(* CoDeSys 2.3 project: drillMachine_Simple_Turku.pro *)
(* Title: Use of different IEC-61131-3 languages *)
(* Version: 1.0.0 *)
(* Author: Niko Siltala (TUT) *)
(* Description: Use of different IEC-61131-3 languages to control a lift door. *)
(* Libraries: Util.lib 16.8.17 14:08:57, STANDARD.LIB 16.8.17 14:08:57 *)

(* Global variable list: Global_Variables *)
VAR_GLOBAL
	(*ConveyourIn - Left*)
	I_ConvIn_PartPresent: BOOL;	(*Sensor: Part is present*)
	O_ConvIn_MotON		: BOOL;	(*Conveyour In: Motor ON*)

	(*ConveyourOut - Right*)
	I_ConvOut_PartPresent: BOOL;(*Sensor: Part is present*)
	O_ConvOut_MotON		: BOOL;	(*Conveyour Out: Motor ON*)

	(*Manipulator - Left*)
	I_ManiL_Limit_Up	: BOOL;	(*Manipulator Left: Limit: Up*)
	I_ManiL_Limit_Dn	: BOOL;	(*Manipulator Left: Limit: Down*)
	I_ManiL_Limit_Home	: BOOL;	(*Manipulator Left: Home sensor*)
	I_ManiL_Turned_Left	: BOOL;	(*Manipulator Left: Turned to left*)
	I_ManiL_Turned_Right: BOOL;	(*Manipulator Left: Turned to right*)
	I_ManiL_Gripper_Open: BOOL;	(*Manipulator Left: Gripper is open*)

	O_ManiL_Turn_Left	: BOOL;	(*Manipulator Left: Turn to left position. Controls the valve*)
	O_ManiL_Turn_Right	: BOOL;	(*Manipulator Left: Turn to right position. Controls the valve*)
	O_ManiL_Gripper_Close: BOOL;(*Manipulator Left: Closes Gripper. Controls the valve*)

	bManiL_axZ_Enable	: BOOL;	(*Manipulator Left: Z-axis: enable*)
	bManiL_axZ_Start	: BOOL;	(*Manipulator Left: Z-axis: Start motion*)
	fManiL_axZ_Velo		: REAL;	(*Manipulator Left: Z-axis: Velocity*)
	fManiL_axZ_TargetPos: REAL;	(*Manipulator Left: Z-axis: Target position*)
	fManiL_axZ_CurrPos	: REAL;	(*Manipulator Left: Z-axis: Current position*)
	bManiL_axZ_InTargetPos	: BOOL;	(*Manipulator Left: Z-axis: Target position is reached*)

	(*Drilling Machine*)
	I_Drill_Limit_Up	: BOOL;	(*Drill: Limit: Up*)
	I_Drill_Limit_Dn	: BOOL;	(*Drill: Limit: Down*)
	I_Drill_Limit_Home	: BOOL;	(*Drill: Home sensor*)
	I_Drill_Fixture_Open: BOOL;	(*Drill: Fixture is open*)
	I_Drill_Fixture_Closed: BOOL;	(*Drill: Fixture is closed*)

	O_Drill_Spindle_On	: BOOL;	(*Drill: Turn on drill spindle.*)
	O_Drill_Fixture_Close: BOOL;(*Drill: Closes Fixture. Controls the valve*)

	bDrill_axZ_Enable	: BOOL;	(*Drill: Z-axis: enable*)
	bDrill_axZ_Start	: BOOL;	(*Drill: Z-axis: Start motion*)
	fDrill_axZ_Velo		: REAL;	(*Drill: Z-axis: Velocity*)
	fDrill_axZ_TargetPos: REAL;	(*Drill: Z-axis: Target position*)
	fDrill_axZ_CurrPos	: REAL;	(*Drill: Z-axis: Current position*)
	bDrill_axZ_InTargetPos	: BOOL;	(*Drill: Z-axis: Target position is reached*)

	(*Manipulator - Right*)
	I_ManiR_Limit_Up	: BOOL;	(*Manipulator Right: Limit: Up*)
	I_ManiR_Limit_Dn	: BOOL;	(*Manipulator Right: Limit: Down*)
	I_ManiR_Limit_Home	: BOOL;	(*Manipulator Right: Home sensor*)
	I_ManiR_Turned_Left	: BOOL;	(*Manipulator Right: Turned to left*)
	I_ManiR_Turned_Right: BOOL;	(*Manipulator Right: Turned to right*)
	I_ManiR_Gripper_Open: BOOL;	(*Manipulator Right: Gripper is open*)

	O_ManiR_Turn_Left	: BOOL;	(*Manipulator Right: Turn to left position. Controls the valve*)
	O_ManiR_Turn_Right	: BOOL;	(*Manipulator Right: Turn to right position. Controls the valve*)
	O_ManiR_Gripper_Close: BOOL;(*Manipulator Right: Closes Gripper. Controls the valve*)

	bManiR_axZ_Enable	: BOOL;	(*Manipulator Right: Z-axis: enable*)
	bManiR_axZ_Start	: BOOL;	(*Manipulator Right: Z-axis: Start motion*)
	fManiR_axZ_Velo		: REAL;	(*Manipulator Right: Z-axis: Velocity*)
	fManiR_axZ_TargetPos: REAL;	(*Manipulator Right: Z-axis: Target position*)
	fManiR_axZ_CurrPos	: REAL;	(*Manipulator Right: Z-axis: Current position*)
	bManiR_axZ_InTargetPos	: BOOL;	(*Manipulator Right: Z-axis: Target position is reached*)


	(*Control panel and indications*)
	I_EmergencyClear	: BOOL;	(*Emergency Circuit is clear*)
	I_Btn_Reset		: BOOL;	(*Button: Reset*)
	I_Btn_Start		: BOOL;	(*Button: Start*)
	I_Btn_Stop		: BOOL;	(*Button: Stop*)
	I_Btn_CycleStart: BOOL;	(*Button: Cycle Start*)

	O_Light_Running	: BOOL;	(*Light: Running*)
	O_Light_Stopped	: BOOL;	(*Light: Stopped*)
	O_Beacon_Red	: BOOL;	(*Beacon Light: red*)
	O_Beacon_Yellow	: BOOL;	(*Beacon Light: yellow*)
	O_Beacon_Green	: BOOL;	(*Beacon Light: green*)

END_VAR

(* Data type *)
TYPE ST_Part :
(*Data structure for the simulated parts *)
STRUCT
	bExists		: BOOL;	(* Part exists *)
	bHasHole	: BOOL;	(* Part has hole *)
	posX		: REAL;	(* X-position of the part*)
	posY		: REAL;	(* Y-position of the part*)
END_STRUCT
END_TYPE

(* POU PRG_MAIN, ST *)
PROGRAM PRG_MAIN
VAR
	fbSFCExample : FB_SFC_Example;
END_VAR
(*START MAKING YOUR DRILLING SYSTEM PROGRAM HERE*)
fbSFCExample();
PRG_SFCDrilling(bReset:= );
END_PROGRAM

(* POU Examples/FB_SFC_Example, SFC *)
FUNCTION_BLOCK FB_SFC_Example
VAR_INPUT
	bReset		: BOOL;	(*Reset Request*)
END_VAR
VAR_OUTPUT
END_VAR
VAR
	bLocalReset	: BOOL;	(*Performs local reset*)
	SFCReset 	: BOOL;	(*Resets the execution of SFC to init once this SFCFlag is set true *)
END_VAR
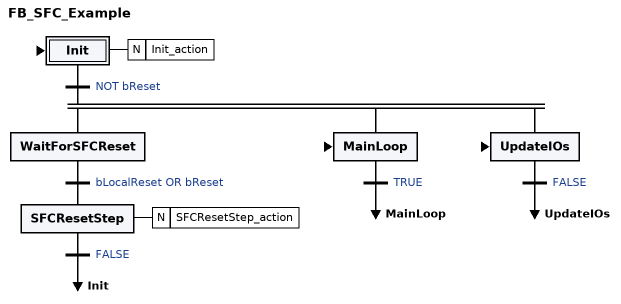
INITIAL_STEP Init:
	Init_action(N);
END_STEP
TRANSITION FROM Init TO (WaitForSFCReset, MainLoop, UpdateIOs) := NOT bReset;
END_TRANSITION
STEP WaitForSFCReset:
END_STEP
TRANSITION FROM WaitForSFCReset TO SFCResetStep := bLocalReset OR bReset;
END_TRANSITION
STEP SFCResetStep:
	SFCResetStep_action(N);
END_STEP
TRANSITION FROM SFCResetStep TO Init := FALSE;
END_TRANSITION
STEP MainLoop:
END_STEP
TRANSITION FROM MainLoop TO MainLoop := TRUE;
END_TRANSITION
STEP UpdateIOs:
END_STEP
TRANSITION FROM UpdateIOs TO UpdateIOs := FALSE;
END_TRANSITION

ACTION Init_action:
SFCReset := FALSE;
bLocalReset	:= FALSE;
END_ACTION

ACTION SFCResetStep_action:
SFCReset := TRUE;
END_ACTION
END_FUNCTION_BLOCK

(* POU PRG_SFCDrilling, SFC *)
PROGRAM PRG_SFCDrilling
VAR_INPUT
	bReset		: BOOL;	(*Reset Request*)
END_VAR
VAR_OUTPUT
END_VAR
VAR
	bLocalReset	: BOOL;	(*Performs local reset*)
	SFCReset 	: BOOL;	(*Resets the execution of SFC to init once this SFCFlag is set true *)
	tonViive	: TON;		(*Liikkeen monitoroinnin viive*)
	tStartDelay: TIME := T#1s;
END_VAR
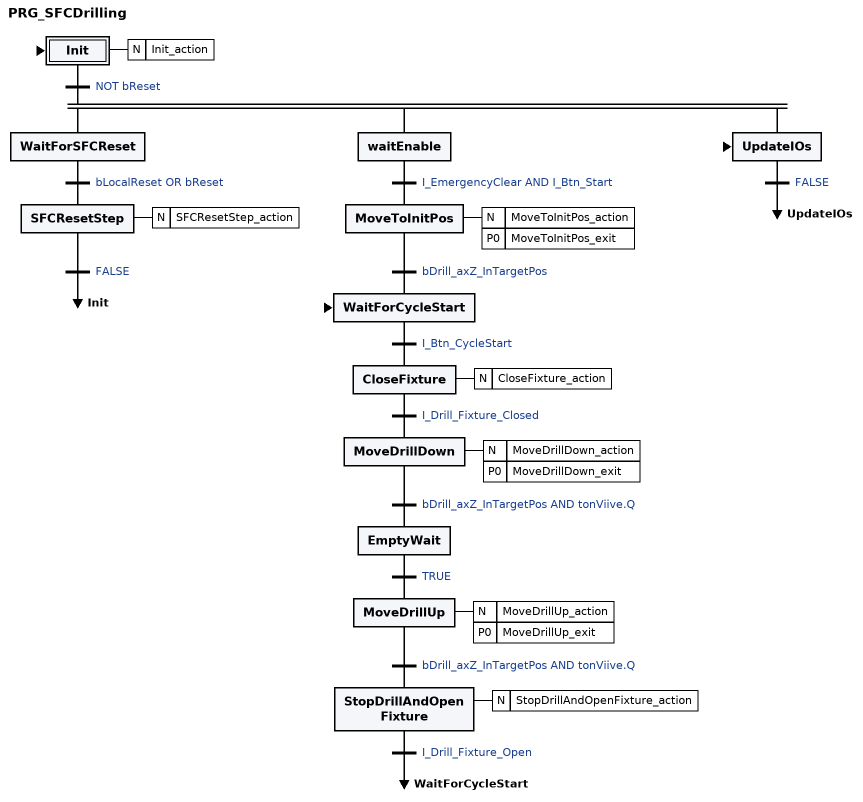
INITIAL_STEP Init:
	Init_action(N);
END_STEP
TRANSITION FROM Init TO (WaitForSFCReset, waitEnable, UpdateIOs) := NOT bReset;
END_TRANSITION
STEP WaitForSFCReset:
END_STEP
TRANSITION FROM WaitForSFCReset TO SFCResetStep := bLocalReset OR bReset;
END_TRANSITION
STEP SFCResetStep:
	SFCResetStep_action(N);
END_STEP
TRANSITION FROM SFCResetStep TO Init := FALSE;
END_TRANSITION
STEP waitEnable:
END_STEP
TRANSITION FROM waitEnable TO MoveToInitPos := I_EmergencyClear AND I_Btn_Start;
END_TRANSITION
STEP MoveToInitPos:
	MoveToInitPos_action(N);
	MoveToInitPos_exit(P0);
END_STEP
TRANSITION FROM MoveToInitPos TO WaitForCycleStart := bDrill_axZ_InTargetPos;
END_TRANSITION
STEP WaitForCycleStart:
END_STEP
TRANSITION FROM WaitForCycleStart TO CloseFixture := I_Btn_CycleStart;
END_TRANSITION
STEP CloseFixture:
	CloseFixture_action(N);
END_STEP
TRANSITION FROM CloseFixture TO MoveDrillDown := I_Drill_Fixture_Closed;
END_TRANSITION
STEP MoveDrillDown:
	MoveDrillDown_action(N);
	MoveDrillDown_exit(P0);
END_STEP
TRANSITION FROM MoveDrillDown TO EmptyWait := bDrill_axZ_InTargetPos AND tonViive.Q;
END_TRANSITION
STEP EmptyWait:
END_STEP
TRANSITION FROM EmptyWait TO MoveDrillUp := TRUE;
END_TRANSITION
STEP MoveDrillUp:
	MoveDrillUp_action(N);
	MoveDrillUp_exit(P0);
END_STEP
TRANSITION FROM MoveDrillUp TO StopDrillAndOpenFixture := bDrill_axZ_InTargetPos AND tonViive.Q;
END_TRANSITION
STEP StopDrillAndOpenFixture:
	StopDrillAndOpenFixture_action(N);
END_STEP
TRANSITION FROM StopDrillAndOpenFixture TO WaitForCycleStart := I_Drill_Fixture_Open;
END_TRANSITION
STEP UpdateIOs:
END_STEP
TRANSITION FROM UpdateIOs TO UpdateIOs := FALSE;
END_TRANSITION

ACTION Init_action:
SFCReset := FALSE;
bLocalReset	:= FALSE;
END_ACTION

ACTION SFCResetStep_action:
SFCReset := TRUE;
END_ACTION

ACTION MoveToInitPos_action:
bDrill_axZ_Enable := TRUE;
fDrill_axZ_Velo := 5;
fDrill_axZ_TargetPos := -10;
bDrill_axZ_Start := TRUE;
END_ACTION

ACTION MoveToInitPos_exit:
bDrill_axZ_Start := FALSE;
END_ACTION

ACTION CloseFixture_action:
O_Drill_Fixture_Close := TRUE;
END_ACTION

ACTION MoveDrillDown_action:
fDrill_axZ_Velo :=10;
fDrill_axZ_TargetPos := -140;
bDrill_axZ_Start := TRUE;
tonViive(IN:=TRUE , PT:= tStartDelay);
O_Drill_Spindle_On := TRUE;
END_ACTION

ACTION MoveDrillDown_exit:
bDrill_axZ_Start := FALSE;
tonViive(IN:=FALSE );
END_ACTION

ACTION MoveDrillUp_action:
fDrill_axZ_TargetPos := -10;
bDrill_axZ_Start := TRUE;
tonViive(IN:=TRUE , PT:= tStartDelay);
END_ACTION

ACTION MoveDrillUp_exit:
bDrill_axZ_Start := FALSE;
tonViive(IN:=FALSE );
END_ACTION

ACTION StopDrillAndOpenFixture_action:
O_Drill_Spindle_On := FALSE;
O_Drill_Fixture_Close := FALSE;
END_ACTION
END_PROGRAM

(* POU Examples/PRG_SFC_Example, SFC *)
PROGRAM PRG_SFC_Example
VAR_INPUT
	bReset		: BOOL;	(*Reset Request*)
END_VAR
VAR_OUTPUT
END_VAR
VAR
	bLocalReset	: BOOL;	(*Performs local reset*)
	SFCReset 	: BOOL;	(*Resets the execution of SFC to init once this SFCFlag is set true *)
END_VAR
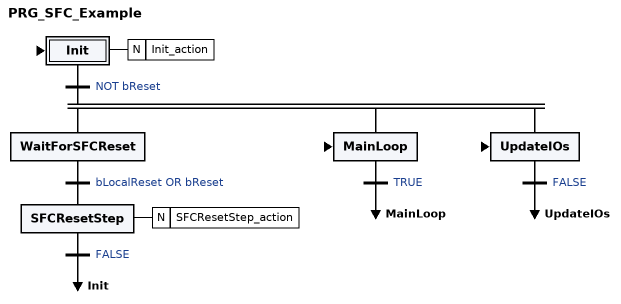
INITIAL_STEP Init:
	Init_action(N);
END_STEP
TRANSITION FROM Init TO (WaitForSFCReset, MainLoop, UpdateIOs) := NOT bReset;
END_TRANSITION
STEP WaitForSFCReset:
END_STEP
TRANSITION FROM WaitForSFCReset TO SFCResetStep := bLocalReset OR bReset;
END_TRANSITION
STEP SFCResetStep:
	SFCResetStep_action(N);
END_STEP
TRANSITION FROM SFCResetStep TO Init := FALSE;
END_TRANSITION
STEP MainLoop:
END_STEP
TRANSITION FROM MainLoop TO MainLoop := TRUE;
END_TRANSITION
STEP UpdateIOs:
END_STEP
TRANSITION FROM UpdateIOs TO UpdateIOs := FALSE;
END_TRANSITION

ACTION Init_action:
SFCReset := FALSE;
bLocalReset	:= FALSE;
END_ACTION

ACTION SFCResetStep_action:
SFCReset := TRUE;
END_ACTION
END_PROGRAM

(* POU Simulation/PRG_Simulator, ST *)
PROGRAM PRG_Simulator
(*This Program is simulating the real machine and mimics its behaviour.
The main task is to update the inputs for students program according the stimulus student provides as outputs.
Another task is to monitor (physical) error conditions occuring in the system and record them.
Author: Niko Siltala, niko.siltala@tut.fi, Tampere University of Technology / MEI
Date: 2016-12-12
Version: 1.0
*) 
VAR
	bBtn_EmergencyStop	: BOOL;	(*Emergency Stop button*)
	rsEmergencyClear	: RS;	(*RS - flip-flop for Emergency clear info*)
	i 	: INT;
	c 	: INT;
	fbManipLeft		: FB_Simu_Manipulator;	(*Left simulated manipulator *)
	fbManipRight	: FB_Simu_Manipulator;	(*Right simulated manipulator *)
	fbDrill			: FB_Simu_Drill;		(*Drill machine simulated*)
	arrParts_ConvIn		: ARRAY [0..10] OF ST_Part; (*Parts on input conveyour*)
	arrParts_ConvOut	: ARRAY [0..10] OF ST_Part; (*Parts on output conveyour*)
	stPart_inMLeftGripper 	: ST_Part; 	(*Data structure for the part*)
	stPart_inMRightGripper 	: ST_Part; 	(*Data structure for the part*)
	stPart_inDrillFixture 	: ST_Part; 	(*Data structure for the part*)
	bAddPartOnConvIn		: BOOL;	(*Adds new part on conveyor*)
	bAddPartInDrill			: BOOL;	(*Adds new part into drilling machine*)
	bRemovePartFromDrill	: BOOL;	(*Adds new part into drilling machine*)
	bClearErrors			: BOOL;	(*Clear Errors*)
	bClearSystem			: BOOL;	(*Clears system from parts *)
	RT_AddPart				: R_TRIG;
	RT_RemovePart			: R_TRIG;
	wError_ManipL			: WORD;	(*Error bits between convIn and Manip_Left*)
	wError_Drill			: WORD; (*Error bits at drill*)
	wError_ManipR			: WORD;	(*Error bits between convIn and Manip_Left*)
	iState_IF				: ARRAY [1..5] OF UINT;	(*State variable; Exchange between 1=ConvIn->ManipL, 2=ManipL->Drill, 3=Drill->ManipR, 4=ManipR->ConvOut, 5=Drill*)
END_VAR
VAR CONSTANT
	bMANUAL_CONTROLS				: BOOL 	:=FALSE;(*Manual override for controls*)
	fPOS_MANIP_CONV_NO_PART_SAFE	: REAL	:= 90;	(*Manipulator on conv with NO part - Safe to move*)
	fPOS_MANIP_CONV_WITH_PART_SAFE	: REAL	:= 70;	(*Manipulator on conv with part - Safe to move*)
	fPOS_MANIP_CONV_PICK_LEVEL		: REAL	:= 120;	(*Manipulator Pick/place level on conv*)
	fPOS_MANIP_DRILL_WITH_PART_SAFE	: REAL	:= 53;	(*Manipulator coming to drill with part - Safe to move*)
	fPOS_MANIP_DRILL_NO_PART_SAFE	: REAL	:= 46;	(*Manipulator coming to drill with NO part - Safe to move*)
	fPOS_MANIP_DRILL_PICK_LEVEL		: REAL	:= 74;	(*Manipulator Pick/place level on Drill*)
	fPOS_MANIP_PICK_TOLERANCE		: REAL	:= 30;	(*Manipulator Pick level tolerance from the part (=fingers length)*)
	fPART_HEIGH						: REAL	:= 50;	(*Part height*)
	fPART_PICK_TOLERANCE			: REAL	:= 10;	(*Part pick & place (negative) tolerance from Levels.*)
	fPART_HOLE_DEPTH_REQ			: REAL	:= 40;	(*Part required Hole depth*)
	fPART_HOLE_DEPTH_MAX			: REAL	:= 45;	(*Max Hole depth*)
	fPOS_DRILL_BIT_TOUCHES			: REAL	:= 100;	(*Drill touches the part*)
	iDRILL_SPINDLE_MIN_FOR_DRILLING	: INT	:= 400;	(*Minimum spindle speed for drilling*)
END_VAR
(*Handle counter*)
c:= c+1;
IF c> 10 THEN
	c:= 0;
END_IF;

(*Simulate emergency stop circuitry*)
rsEmergencyClear(
	SET:= I_Btn_Reset,
	RESET1:= bBtn_EmergencyStop,
	Q1=> I_EmergencyClear);

(*Adds new part into drill fixture*)
RT_AddPart(CLK:=bAddPartInDrill , Q=> );
IF RT_AddPart.Q AND NOT stPart_inDrillFixture.bExists THEN
	IF fbDrill.bFixture_Closed THEN
		(*Part inserted when the fixture is closed*)
		wError_Drill.4 := TRUE;	(*Fixture closed when inserting part*)
	ELSE
		(*Part inserted to fixture*)
		stPart_inDrillFixture.bExists := TRUE;
		stPart_inDrillFixture.bHasHole := FALSE;
	END_IF;
END_IF;

(*Remove part from drill fixture*)
RT_RemovePart(CLK:=bRemovePartFromDrill , Q=> );
IF RT_RemovePart.Q AND stPart_inDrillFixture.bExists THEN
	IF fbDrill.bFixture_Closed THEN
		(*Part removed when the fixture is closed*)
		wError_Drill.5 := TRUE;	(*Fixture closed while leaving with part*)
	ELSE
		(*Part removed*)
		stPart_inDrillFixture.bExists := FALSE;
	END_IF;
END_IF;


IF bMANUAL_CONTROLS THEN

	(*Call drill machine*)
	fbDrill(
		bEnable:= ,
		bLift_Start:= ,
		fLift_Velo:= ,
		fLift_TargetPos:= , 
		bDrillOn:= , 
		bFixture_Close:= , 
		stPart_inFixture:= stPart_inDrillFixture,
		bLift_InTarget=> bDrill_axZ_InTargetPos,
		fLift_CurrentPos=> fDrill_axZ_CurrPos,
		bLimit_Top=> I_Drill_Limit_Up,
		bLimit_Bottom=> I_Drill_Limit_Dn,
		bHome_Sensor=> I_Drill_Limit_Home,
		bFixture_Open=> I_Drill_Fixture_Open,
		bFixture_Closed=> I_Drill_Fixture_Closed);

ELSE

	(*Call drill machine*)
	fbDrill(
		bEnable:= bDrill_axZ_Enable,
		bLift_Start:= bDrill_axZ_Start,
		fLift_Velo:= fDrill_axZ_Velo,
		fLift_TargetPos:= fDrill_axZ_TargetPos,
		bDrillOn:= O_Drill_Spindle_On,
		bFixture_Close:= O_Drill_Fixture_Close,
		stPart_inFixture:= stPart_inDrillFixture,
		bLift_InTarget=> bDrill_axZ_InTargetPos,
		fLift_CurrentPos=> fDrill_axZ_CurrPos,
		bLimit_Top=> I_Drill_Limit_Up,
		bLimit_Bottom=> I_Drill_Limit_Dn,
		bHome_Sensor=> I_Drill_Limit_Home,
		bFixture_Open=> I_Drill_Fixture_Open,
		bFixture_Closed=> I_Drill_Fixture_Closed);
END_IF;


(*Make drilling and check error conditions at Drilling*)
ErrorCheck_Drill;


(*Clear active errors*)
IF bClearErrors THEN
	wError_ManipL := 0;
	wError_Drill := 0;
	wError_ManipR := 0;
END_IF;

(*Remove parts from entire system*)
IF bClearSystem THEN
	(*Clear input & output conveyour from parts*)
	FOR i:= 0 TO 10 DO
		arrParts_ConvIn[i].bExists := FALSE;
		arrParts_ConvOut[i].bExists := FALSE;
	END_FOR;
	(*Clear Manipulators and drill from parts*)
	stPart_inMLeftGripper.bExists := FALSE;
	stPart_inDrillFixture.bExists := FALSE;
	stPart_inMRightGripper.bExists := FALSE;
END_IF;
END_PROGRAM
ACTION ErrorCheck_Collisions:
(*ManipL and Conveyor collision*)
IF (fbManipLeft.fPos_Y > 140) AND (fbManipLeft.fPos_angle < 50) THEN
	wError_ManipL.7 := TRUE;	(*collision with conveyor*)
END_IF;

(*ManipL and Drill collision*)
IF ((fbDrill.fPos_Y + 16) > fbManipLeft.fPos_Y) AND fbManipLeft.fPos_angle > 150 THEN
	wError_ManipL.1 := TRUE;
	wError_Drill.0 := TRUE;
END_IF;

(*ManipR and Drill collision*)
IF ((fbDrill.fPos_Y + 16) > fbManipRight.fPos_Y) AND fbManipRight.fPos_angle < 50 THEN
	wError_ManipR.1 := TRUE;
	wError_Drill.1 := TRUE;
END_IF;

(*ManipR and Conveyor collision*)
IF (fbManipRight.fPos_Y > 140) AND (fbManipRight.fPos_angle > 150) THEN
	wError_ManipR.7 := TRUE;	(*collision with conveyor*)
END_IF;

(*ManipL and ManipR collision*)
IF (fbManipLeft.fPos_angle > 130) AND (fbManipRight.fPos_angle < 50) AND
  (ABS(fbManipRight.fPos_Y - fbManipLeft.fPos_Y) < 60) THEN
	wError_ManipL.9 := TRUE;	(*collision sidewise with ManipulatorRight*)
	wError_ManipR.9 := TRUE;	(*collision sidewise with ManipulatorLeft*)
END_IF;
END_ACTION
ACTION ErrorCheck_Drill:
(*State model for Drilling.
Includes all associated error conditions and judgements *)

(*Resetting errorCheck*)
IF bClearErrors THEN
	iState_IF[5] := 0;
END_IF;

(*Drilling cycle has been initiated, but part is removed somewhere between.*)
IF (iState_IF[5] > 0) AND NOT stPart_inDrillFixture.bExists THEN
	iState_IF[5] := 0;
END_IF;

(*Drilled too long*)
IF stPart_inDrillFixture.bExists AND
  (fbDrill.fPos_Y > (fPOS_DRILL_BIT_TOUCHES + fPART_HOLE_DEPTH_MAX)) THEN
	wError_Drill.2 := TRUE;	(*collision with part and Drill*)
END_IF;


CASE iState_IF[5] OF
0: (* IDLE *)
	IF fbDrill.fPos_Y > ( fPOS_DRILL_BIT_TOUCHES - fPART_HEIGH ) THEN
		iState_IF[5] := 1;
	END_IF;

1: (* Approaches with Drill *)
	IF  fbDrill.fPos_Y >= fPOS_DRILL_BIT_TOUCHES THEN
		iState_IF[5] := 2;
	END_IF;

2: (* Drilling *)
	IF fbDrill.fPos_Y >= (fPOS_DRILL_BIT_TOUCHES + fPART_HOLE_DEPTH_REQ ) THEN
		iState_IF[5] := 3;
	END_IF;
	IF stPart_inDrillFixture.bExists AND NOT fbDrill.bFixture_Closed THEN
		wError_Drill.7 := TRUE;	(*Drilling without closed fixture*)
	END_IF;
	IF stPart_inDrillFixture.bExists AND fbDrill.iRPMCurrent < iDRILL_SPINDLE_MIN_FOR_DRILLING THEN
		wError_Drill.2 := TRUE;	(*collision with part and Drill*)
		wError_Drill.6 := TRUE;	(*Drilling without sufficient spindle RPM*)
	END_IF;

3: (* Drilled *)
	stPart_inDrillFixture.bHasHole := TRUE;
	IF fbDrill.fPos_Y < fPOS_DRILL_BIT_TOUCHES THEN
		iState_IF[5] := 4;
	END_IF;

4: (* moved up from part *)
	stPart_inDrillFixture.bHasHole := TRUE;
	IF fbDrill.fPos_Y < 30 THEN
		iState_IF[5] := 5;
	END_IF;

5: (* moved to wait area *)
	iState_IF[5] := 0;

ELSE
	iState_IF[5] := 0;
END_CASE;
END_ACTION
ACTION ErrorCheck_ManipLeft_ConvIn:
(*State model for exchanging part from ConveyorIn to ManipLeft.
Includes all associated error conditions and judgements *)

CASE iState_IF[1] OF
0: (* IDLE *)
	IF arrParts_ConvIn[0].bExists AND NOT stPart_inMLeftGripper.bExists THEN
		iState_IF[1] := 1;
	END_IF;

1: (* waitMoveAbove *)
	IF fbManipLeft.bBeamAtLeft AND fbManipLeft.fPos_Y < fPOS_MANIP_CONV_NO_PART_SAFE THEN
		iState_IF[1] := 2;
	END_IF;
	IF fbManipLeft.fPos_angle < 30 AND fbManipLeft.fPos_Y > fPOS_MANIP_CONV_NO_PART_SAFE THEN
		wError_ManipL.0 := TRUE;
	END_IF;

2: (* ManipulatorLeft is above *)
	IF fbManipLeft.bBeamAtLeft AND fbManipLeft.fPos_Y >= fPOS_MANIP_CONV_NO_PART_SAFE THEN
		iState_IF[1] := 3;
	END_IF;
	IF NOT fbManipLeft.bBeamAtLeft AND fbManipLeft.fPos_angle < 30 AND fbManipLeft.fPos_Y > fPOS_MANIP_CONV_NO_PART_SAFE THEN
		wError_ManipL.0 := TRUE;
	END_IF;

3: (* Approaches from above *)
	IF fbManipLeft.bBeamAtLeft AND fbManipLeft.bGripperIsOpen AND
	  fbManipLeft.fPos_Y >= (fPOS_MANIP_CONV_PICK_LEVEL - 2*fPART_PICK_TOLERANCE) THEN
		iState_IF[1] := 4;
	ELSIF fbManipLeft.fPos_Y < fPOS_MANIP_CONV_NO_PART_SAFE THEN
		iState_IF[1] := 0;
	END_IF;
	IF NOT fbManipLeft.bBeamAtLeft THEN
		wError_ManipL.0 := TRUE;
	END_IF;
	IF NOT fbManipLeft.bGripperIsOpen THEN
		wError_ManipL.5 := TRUE;
	END_IF;

4: (* Over part *)
	IF fbManipLeft.bBeamAtLeft AND fbManipLeft.fPos_Y >= (fPOS_MANIP_CONV_PICK_LEVEL - fPART_PICK_TOLERANCE) AND
	fbManipLeft.fPos_Y <= fPOS_MANIP_CONV_PICK_LEVEL AND fbManipLeft.bGripperClosed THEN
		(*Grasping occurs*)
		iState_IF[1] := 5;
		(*TODO: Add part grasp height compensation*)
	ELSIF fbManipLeft.fPos_Y < fPOS_MANIP_CONV_NO_PART_SAFE THEN
		iState_IF[1] := 0;
	END_IF;
	IF NOT fbManipLeft.bBeamAtLeft THEN
		wError_ManipL.0 := TRUE;
	END_IF;
	IF fbManipLeft.fPos_Y > fPOS_MANIP_CONV_PICK_LEVEL THEN
		wError_ManipL.2 := TRUE;
	END_IF;

5: (* part grasped *)
	stPart_inMLeftGripper.bExists := TRUE;
	IF fbManipLeft.bBeamAtLeft AND fbManipLeft.fPos_Y < fPOS_MANIP_CONV_WITH_PART_SAFE THEN
		iState_IF[1] := 6;
	END_IF;
	IF NOT fbManipLeft.bBeamAtLeft AND fbManipLeft.fPos_Y > fPOS_MANIP_CONV_NO_PART_SAFE THEN
		wError_ManipL.3 := TRUE;
	END_IF;

6: (* moved up with part *)
	IF fbManipLeft.fPos_Y < fPOS_MANIP_CONV_WITH_PART_SAFE THEN
		iState_IF[1] := 7;
	END_IF;

7: (* moved up with part *)
	arrParts_ConvIn[0].bExists := FALSE;
	iState_IF[1] := 0;

ELSE
	iState_IF[1] := 0;
END_CASE;
END_ACTION
ACTION ErrorCheck_ManipLeft_Drill:
(*State model for exchanging part from ManipLeft to Drill.
Includes all associated error conditions and judgements *)

(*Dropping part from gripper too soon*)
IF (iState_IF[2] > 0) AND (iState_IF[2] <= 3) AND NOT fbManipLeft.bGripperClosed THEN
	wError_ManipL.6 := TRUE;
	iState_IF[2] := 0;
END_IF;

(*Collision with parts*)
IF stPart_inMLeftGripper.bExists AND stPart_inDrillFixture.bExists AND fbManipLeft.bBeamAtRight AND
  fbManipLeft.fPos_Y > (fPOS_MANIP_DRILL_PICK_LEVEL - 2* fPART_HEIGH) THEN
	wError_Drill.3 := TRUE;
END_IF;

(*Part exchange sequence*)
CASE iState_IF[2] OF
0: (* IDLE *)
	IF stPart_inMLeftGripper.bExists AND fbManipLeft.bGripperClosed THEN
		iState_IF[2] := 1;
	END_IF;

1: (* waitMoveAbove *)
	IF fbManipLeft.bBeamAtRight AND fbManipLeft.fPos_Y < fPOS_MANIP_DRILL_WITH_PART_SAFE THEN
		iState_IF[2] := 2;
	END_IF;
	IF fbManipLeft.fPos_angle > 150 AND fbManipLeft.fPos_Y > fPOS_MANIP_DRILL_WITH_PART_SAFE THEN
		wError_ManipL.1 := TRUE;
	END_IF;

2: (* ManipulatorLeft is above release point*)
	IF fbManipLeft.bBeamAtRight AND fbManipLeft.fPos_Y >= fPOS_MANIP_DRILL_WITH_PART_SAFE THEN
		iState_IF[2] := 3;
	END_IF;
	IF NOT fbManipLeft.bBeamAtRight AND (fbManipLeft.fPos_angle > 150) AND
	  (fbManipLeft.fPos_Y > fPOS_MANIP_DRILL_WITH_PART_SAFE) THEN
		wError_ManipL.1 := TRUE;
	END_IF;

3: (* Approaches from above *)
	IF fbManipLeft.bBeamAtRight AND fbManipLeft.bGripperClosed AND
	  (fbManipLeft.fPos_Y >= (fPOS_MANIP_DRILL_PICK_LEVEL - fPART_PICK_TOLERANCE)) THEN
		iState_IF[2] := 4;
	ELSIF fbManipLeft.fPos_Y < fPOS_MANIP_DRILL_WITH_PART_SAFE THEN
		iState_IF[2] := 0;
	END_IF;
	IF NOT fbManipLeft.bBeamAtRight AND fbManipLeft.fPos_Y > fPOS_MANIP_DRILL_WITH_PART_SAFE THEN
		wError_ManipL.1 := TRUE;
	END_IF;

4: (* At release point *)
	(*Errors*)
	IF stPart_inDrillFixture.bExists THEN
		wError_ManipL.2 := TRUE;
		wError_Drill.3 := TRUE;
	END_IF;
	(*State trensition*)
	IF fbManipLeft.bBeamAtRight AND (fbManipLeft.fPos_Y >= (fPOS_MANIP_DRILL_PICK_LEVEL - fPART_PICK_TOLERANCE)) AND
	fbManipLeft.fPos_Y <= fPOS_MANIP_DRILL_PICK_LEVEL AND fbManipLeft.bGripperIsOpen THEN
		(*Release occurs*)
		iState_IF[2] := 5;
		(*Copy part to Drill Fixture*)
		F_CopyPart(stPart_inMLeftGripper, stPart_inDrillFixture);
		stPart_inMLeftGripper.bExists := FALSE;
	ELSIF fbManipLeft.fPos_Y < fPOS_MANIP_DRILL_WITH_PART_SAFE THEN
		iState_IF[2] := 0;
	END_IF;
	IF NOT fbManipLeft.bBeamAtRight AND fbManipLeft.fPos_Y > fPOS_MANIP_DRILL_WITH_PART_SAFE THEN
		wError_ManipL.1 := TRUE;
	END_IF;
	IF fbManipLeft.fPos_Y > fPOS_MANIP_DRILL_PICK_LEVEL THEN
		wError_ManipL.2 := TRUE;
	END_IF;
	IF fbDrill.bFixture_Closed THEN
		wError_Drill.4 := TRUE;	(*Fixture closed when inserting part*)
	END_IF;

5: (* Release part *)
	IF fbManipLeft.bBeamAtRight AND fbManipLeft.fPos_Y <= fPOS_MANIP_DRILL_NO_PART_SAFE THEN
		iState_IF[2] := 6;
	ELSIF fbManipLeft.bBeamAtLeft AND fbManipLeft.fPos_Y <= fPOS_MANIP_CONV_NO_PART_SAFE THEN
		(* Errornous leave condition*)
		iState_IF[2] := 0;
	END_IF;
	IF NOT fbManipLeft.bBeamAtRight AND fbManipLeft.fPos_Y > fPOS_MANIP_DRILL_NO_PART_SAFE THEN
		wError_ManipL.1 := TRUE;
		wError_ManipL.3 := TRUE;
	END_IF;
	IF NOT fbManipLeft.bGripperIsOpen THEN
		wError_ManipR.10 := TRUE;	(*re-grasping released part*)
	END_IF;

6: (* moved up *)
	IF fbManipLeft.fPos_Y <= fPOS_MANIP_DRILL_NO_PART_SAFE THEN
		iState_IF[2] := 7;
	END_IF;
	iState_IF[2] := 0;

7: (* Can move away *)
	iState_IF[2] := 0;

ELSE
	iState_IF[2] := 0;
END_CASE;
END_ACTION
ACTION ErrorCheck_ManipRight_ConvOut:
(*State model for exchanging part from ManipRight to Conveyor.
Includes all associated error conditions and judgements *)

(*Dropping part from gripper too soon*)
IF (iState_IF[4] > 0) AND (iState_IF[4] <= 3) AND NOT fbManipRight.bGripperClosed THEN
	wError_ManipR.6 := TRUE;
	iState_IF[4] := 0;
END_IF;

(*Collision with parts*)
IF stPart_inMRightGripper.bExists AND arrParts_ConvOut[5].bExists AND fbManipRight.fPos_angle > 150 AND
  fbManipRight.fPos_Y > (fPOS_MANIP_CONV_PICK_LEVEL - fPART_HEIGH) THEN
	wError_ManipR.8 := TRUE;
END_IF;

(*Part exchange sequence*)
CASE iState_IF[4] OF
0: (* IDLE *)
	IF stPart_inMRightGripper.bExists AND fbManipRight.bGripperClosed THEN
		iState_IF[4] := 1;
	END_IF;

1: (* waitMoveAbove *)
	IF fbManipRight.bBeamAtRight AND fbManipRight.fPos_Y <= fPOS_MANIP_CONV_WITH_PART_SAFE THEN
		iState_IF[4] := 2;
	END_IF;
	IF fbManipRight.fPos_angle > 150 AND fbManipRight.fPos_Y > fPOS_MANIP_CONV_WITH_PART_SAFE THEN
		wError_ManipR.0 := TRUE;
	END_IF;

2: (* ManipulatorRight is above release point*)
	IF fbManipRight.bBeamAtRight AND fbManipRight.fPos_Y >= fPOS_MANIP_CONV_WITH_PART_SAFE THEN
		iState_IF[4] := 3;
	END_IF;
	IF NOT fbManipRight.bBeamAtRight AND (fbManipRight.fPos_angle > 150) AND
	  (fbManipRight.fPos_Y > fPOS_MANIP_CONV_WITH_PART_SAFE) THEN
		wError_ManipR.0 := TRUE;
	END_IF;

3: (* Approaches from above *)
	IF fbManipRight.bBeamAtRight AND fbManipRight.bGripperClosed AND
	  (fbManipRight.fPos_Y >= (fPOS_MANIP_CONV_PICK_LEVEL - fPART_PICK_TOLERANCE)) THEN
		iState_IF[4] := 4;
	ELSIF fbManipRight.fPos_Y < fPOS_MANIP_CONV_WITH_PART_SAFE THEN
		iState_IF[4] := 0;
	END_IF;
	IF NOT fbManipRight.bBeamAtRight AND fbManipRight.fPos_Y > fPOS_MANIP_CONV_WITH_PART_SAFE THEN
		wError_ManipR.0 := TRUE;
	END_IF;

4: (* At release point *)
	(*Errors*)
	IF arrParts_ConvOut[5].bExists THEN
		wError_ManipR.2 := TRUE;
	END_IF;
	(*State trensition*)
	IF fbManipRight.bBeamAtRight AND (fbManipRight.fPos_Y >= (fPOS_MANIP_CONV_PICK_LEVEL - fPART_PICK_TOLERANCE)) AND
	fbManipRight.fPos_Y <= fPOS_MANIP_CONV_PICK_LEVEL AND fbManipRight.bGripperIsOpen THEN
		(*Release occurs*)
		iState_IF[4] := 5;
		(*Copy part to Conveyour Out*)
		F_CopyPart(stPart_inMRightGripper, arrParts_ConvOut[5]);
		(*TODO: Add part grasp height compensation*)
	ELSIF fbManipRight.fPos_Y < fPOS_MANIP_CONV_WITH_PART_SAFE THEN
		iState_IF[4] := 0;
	END_IF;
	IF NOT fbManipRight.bBeamAtRight AND fbManipRight.fPos_Y > fPOS_MANIP_CONV_WITH_PART_SAFE THEN
		wError_ManipR.1 := TRUE;
	END_IF;
	IF fbManipRight.fPos_Y > fPOS_MANIP_CONV_PICK_LEVEL THEN
		wError_ManipR.2 := TRUE;
	END_IF;

5: (* Release part *)
	stPart_inMRightGripper.bExists := FALSE;
	IF fbManipRight.bBeamAtRight AND fbManipRight.fPos_Y <= fPOS_MANIP_CONV_NO_PART_SAFE AND
	   fbManipRight.bGripperIsOpen THEN
		iState_IF[4] := 6;
	END_IF;
	IF NOT fbManipRight.bBeamAtRight AND fbManipRight.fPos_Y > fPOS_MANIP_CONV_NO_PART_SAFE THEN
		wError_ManipR.1 := TRUE;
		wError_ManipR.3 := TRUE;
	END_IF;
	IF NOT fbManipRight.bGripperIsOpen THEN
		wError_ManipR.10 := TRUE;	(*re-grasping released part*)
	END_IF;

6: (* moved up *)
	iState_IF[4] := 0;

ELSE
	iState_IF[4] := 0;
END_CASE;
END_ACTION
ACTION ErrorCheck_ManipRight_Drill:
(*State model for exchanging part from Drive to ManipRight.
Includes all associated error conditions and judgements *)

CASE iState_IF[3] OF
0: (* IDLE *)
	IF stPart_inDrillFixture.bExists AND NOT stPart_inMRightGripper.bExists THEN
		iState_IF[3] := 1;
	END_IF;

1: (* waitMoveAbove *)
	IF fbManipRight.bBeamAtLeft AND fbManipRight.fPos_Y <= fPOS_MANIP_DRILL_NO_PART_SAFE THEN
		iState_IF[3] := 2;
	END_IF;
	IF fbManipRight.fPos_angle < 30 AND fbManipRight.fPos_Y > fPOS_MANIP_DRILL_NO_PART_SAFE THEN
		wError_ManipR.1 := TRUE;
	END_IF;

2: (* ManipulatorLeft is above *)
	IF fbManipRight.bBeamAtLeft AND fbManipRight.fPos_Y >= fPOS_MANIP_DRILL_NO_PART_SAFE THEN
		iState_IF[3] := 3;
	END_IF;
	IF NOT fbManipRight.bBeamAtLeft AND fbManipRight.fPos_angle > 30 AND fbManipRight.fPos_Y > fPOS_MANIP_DRILL_NO_PART_SAFE THEN
		wError_ManipR.1 := TRUE;
	END_IF;

3: (* Approaches from above *)
	IF fbManipRight.bBeamAtLeft AND fbManipRight.bGripperIsOpen AND
	  fbManipRight.fPos_Y >= (fPOS_MANIP_DRILL_PICK_LEVEL - fPART_PICK_TOLERANCE) THEN
		iState_IF[3] := 4;
	ELSIF fbManipRight.fPos_Y < fPOS_MANIP_DRILL_NO_PART_SAFE THEN
		iState_IF[3] := 0;
	END_IF;
	IF NOT fbManipRight.bBeamAtLeft THEN
		wError_ManipR.1 := TRUE;
	END_IF;
	IF NOT fbManipRight.bGripperIsOpen THEN
		wError_ManipR.5 := TRUE;
	END_IF;

4: (* Over part *)
	IF fbManipRight.bBeamAtLeft AND fbManipRight.fPos_Y >= (fPOS_MANIP_DRILL_PICK_LEVEL - fPART_PICK_TOLERANCE) AND
	fbManipRight.fPos_Y <= fPOS_MANIP_DRILL_PICK_LEVEL AND fbManipRight.bGripperClosed THEN
		(*Grasping occurs*)
		iState_IF[3] := 5;
		(*Copy part from Drill Fixture*)
		F_CopyPart(stPart_inDrillFixture, stPart_inMRightGripper);
		(*TODO: Add part grasp height compensation*)
		stPart_inDrillFixture.bExists := FALSE;
		stPart_inDrillFixture.bHasHole := FALSE;
	ELSIF fbManipRight.fPos_Y < fPOS_MANIP_DRILL_NO_PART_SAFE THEN
		iState_IF[3] := 0;
	END_IF;
	IF NOT fbManipRight.bBeamAtLeft THEN
		wError_ManipR.1 := TRUE;
	END_IF;
	IF fbManipRight.fPos_Y > fPOS_MANIP_DRILL_PICK_LEVEL THEN
		wError_ManipR.2 := TRUE;
	END_IF;

5: (* part grasped *)
	IF fbManipRight.bBeamAtLeft AND fbManipRight.fPos_Y < (fPOS_MANIP_DRILL_PICK_LEVEL - fPART_PICK_TOLERANCE) THEN
		iState_IF[3] := 6;
	END_IF;
	IF NOT fbManipRight.bBeamAtLeft AND fbManipRight.fPos_Y > fPOS_MANIP_DRILL_WITH_PART_SAFE THEN
		wError_ManipR.3 := TRUE;
	END_IF;

6: (* leaving with part *)
	IF fbManipRight.bBeamAtLeft AND fbManipRight.fPos_Y <= fPOS_MANIP_DRILL_WITH_PART_SAFE THEN
		iState_IF[3] := 7;
	END_IF;
	IF NOT fbManipRight.bBeamAtLeft AND fbManipRight.fPos_Y > fPOS_MANIP_DRILL_WITH_PART_SAFE THEN
		wError_ManipR.3 := TRUE; 	(*Fixture closed while leaving with part*)
	END_IF;
	IF fbDrill.bFixture_Closed THEN
		wError_Drill.5 := TRUE;	(*Fixture closed while leaving with part*)
	END_IF;

7: (* moved up with part *)
	iState_IF[3] := 0;

ELSE
	iState_IF[3] := 0;
END_CASE;
END_ACTION

(* POU Simulation/FB_Simu_Manipulator, ST *)
FUNCTION_BLOCK FB_Simu_Manipulator
(*Simulation model for the behaviour of the Manipulator.
Author: Niko Siltala, niko.siltala@tut.fi, Tampere University of Technology / MEI
Date: 2016-12-12
Version: 1.0
*)
VAR_INPUT
	bEnable			: BOOL := TRUE;	(*Enable manipulator*)
	bLift_Start		: BOOL;	(*Triggers and starts the lift movement at rising edge*)
	fLift_Velo		: REAL := 10;	(*Velocity*)
	fLift_TargetPos	: REAL;	(*Target position*)
	bBeam_Left		: BOOL;	(*Turn beam at left*)
	bBeam_Right		: BOOL;	(*Turn beam at right*)
	bGripper_Close	: BOOL; (*Close Gripper*)
END_VAR
VAR_OUTPUT
	bGripperIsOpen	: BOOL;	(*Gripper is open*)
	bLift_InTarget	: BOOL;	(*Lift has reached the target*)
	fLift_CurrentPos	: REAL;	(*Current position of the lift*)
	bLimit_Top		: BOOL;	(*Height position at top limit*)
	bLimit_Bottom	: BOOL;	(*Height position at bottom limit*)
	bHome_Sensor	: BOOL;	(*Height position at home limit*)
	bBeamAtRight	: BOOL;	(*Beam turned into right limit*)
	bBeamAtLeft		: BOOL;	(*Beam turned into left limit*)
END_VAR
VAR_IN_OUT
	stPart_inGripper : ST_Part; 	(*Data structure for the part*)
END_VAR
VAR
	fPos_angle	: REAL := 70;	(*Angle of beam [deg]*)
	fPos_height	: REAL;	(* Manipulators height position*)
	fPos_X		: REAL;	(* Manipulator's X position*)
	fPos_Y		: REAL;	(* Manipulator's Y position*)
	fBasePos_Y 	: REAL; (*Position of manipulator base*)
	iState_Lift	: UINT;	(*State of beam model*)
	fPos_Beam_L	: REAL;	(*Beam position left end*)
	fPos_Beam_R	: REAL;	(*Beam position right end*)
	bGripperClosed	: BOOL; (*Gripper is closed*)
	fPosFingerDiff 	: REAL;	(*Right finger position. 0 poistion when grasping.*)
END_VAR
VAR CONSTANT
	iBEAM_LENGTH	: USINT := 120;	(*length of the beam*)
	fPOS_MAX_DOWN	: REAL	:= 220;	(*Max position for down movement*)
END_VAR
(*Simulate axis*)
IF NOT bEnable THEN
	iState_Lift := 0;
END_IF;

CASE iState_Lift OF
0:	(*Off*)
	IF bEnable THEN
		iState_Lift := 1;
	ELSE
		bLift_InTarget := FALSE;
	END_IF;

1:	(*IDLE*)
	IF bLift_Start THEN
		bLift_InTarget := FALSE;
		iState_Lift := 2;
	END_IF;

2:	(*MovingToTarget*)
	bLift_InTarget := FALSE;
	IF fLift_TargetPos > fLift_CurrentPos THEN
		(*Moving up*)
		fLift_CurrentPos := fLift_CurrentPos + ABS(fLift_Velo);
	ELSIF fLift_TargetPos < fLift_CurrentPos THEN
		(*Moving down*)
		fLift_CurrentPos := fLift_CurrentPos - ABS(fLift_Velo);
	END_IF;
	(*Limit output*)
	fLift_CurrentPos := LIMIT(-220, fLift_CurrentPos, 10);
	(* Moved close to target*)
	IF (ABS(fLift_CurrentPos - fLift_TargetPos) <= ABS(fLift_Velo) ) THEN
		fLift_CurrentPos := fLift_TargetPos;
		iState_Lift := 3;
	END_IF;
	(*Start has been removed*)
	IF NOT bLift_Start THEN
		iState_Lift := 1;
	END_IF;

3:	(*In target*)
	bLift_InTarget := TRUE;
	IF NOT bLift_Start THEN
		iState_Lift := 1;
	END_IF;

ELSE	(*Error / to Default*)
	iState_Lift := 0;
END_CASE;

fPos_Y := -fLift_CurrentPos;


(*Simulate Beam turning*)
IF bBeam_Left AND (fPos_angle > 0) AND NOT bBeam_Right THEN
	fPos_angle := LIMIT(0, (fPos_angle - 15), 180);
END_IF;
IF bBeam_Right AND (fPos_angle < 180) AND NOT bBeam_Left THEN
	fPos_angle := LIMIT(0, (fPos_angle + 15), 180);
END_IF;


(*Calculate visualisation positions for lift and beam*)
fPos_X := -iBEAM_LENGTH*COS(3.1415926535897932384626433832795/180*fPos_angle);
(*fPos_Y := fPos_height;*)
fBasePos_Y := fPos_Y;	(*Used for animations as base position*)

(*Calculate endpositions of the visualisation for the beam*)
IF (fPos_X > 0) THEN
	fPos_Beam_L := 0;
	fPos_Beam_R := fPos_X;
ELSE
	fPos_Beam_L := fPos_X;
	fPos_Beam_R := 0;
END_IF;

(*define finger positions*)
IF bGripper_Close THEN
	fPosFingerDiff := 0;
ELSE
	fPosFingerDiff := 10;
END_IF;

(*Set sensor values*)
(*Set output values*)
bLimit_Top := (fPos_Y <= 0);
bLimit_Bottom := (fPos_Y >= 210);
bHome_Sensor := (fPos_Y <= 5) AND (fPos_Y >= -5);

bBeamAtLeft := (fPos_angle <= 0);
bBeamAtRight := (fPos_angle >= 180);

bGripperIsOpen := NOT bGripper_Close;
bGripperClosed := bGripper_Close;
END_FUNCTION_BLOCK

(* POU Simulation/FB_Simu_Drill, ST *)
FUNCTION_BLOCK FB_Simu_Drill
(*Simulation model for the behaviour of the Drill machine.
Author: Niko Siltala, niko.siltala@tut.fi, Tampere University of Technology / MEI
Date: 2016-12-12
Version: 1.0
*)
VAR_INPUT
	bEnable			: BOOL := TRUE;	(*Enable drill*)
	bLift_Start		: BOOL;	(*Triggers and starts the lift movement at rising edge*)
	fLift_Velo		: REAL := 10;	(*Velocity*)
	fLift_TargetPos	: REAL;	(*Target position*)
	bDrillOn		: BOOL;	(*Drill is On*)
	bFixture_Close	: BOOL; (*Close Fixture*)
END_VAR
VAR_OUTPUT
	bLift_InTarget	: BOOL;	(*Lift has reached the target*)
	fLift_CurrentPos	: REAL;	(*Current position of the lift*)
	bLimit_Top		: BOOL;	(*Height position at top limit*)
	bLimit_Bottom	: BOOL;	(*Height position at bottom limit*)
	bHome_Sensor	: BOOL;	(*Height position at home limit*)
	bFixture_Open	: BOOL;	(*Fixture is Open*)
	bFixture_Closed	: BOOL;	(*Fixture is Closed*)
END_VAR
VAR_IN_OUT
	stPart_inFixture : ST_Part; 	(*Data structure for the part*)
END_VAR
VAR
	fPos_height	: REAL;	(* Manipulators height position*)
	fPos_Y		: REAL;	(* Manipulator's Y position*)
	fBasePos_Y 	: REAL; (*Position of manipulator base*)
	iState_Lift	: UINT;	(*State of beam model*)
	iRPMCurrent	: INT;	(*Current RPM*)
	fPosJawDiff 	: REAL;	(*Right fixture jaw position. 0 position when grasping.*)
END_VAR
VAR CONSTANT
	fPOS_MAX_DOWN		: REAL	:= 170;	(*Max position for down movement*)
	iSPINDLE_RPM_MAX	: INT	:= 600;	(*Max RPM for Spindle*)
END_VAR
(*Simulate axis*)
IF NOT bEnable THEN
	iState_Lift := 0;
END_IF;

CASE iState_Lift OF
0:	(*Off*)
	IF bEnable THEN
		iState_Lift := 1;
	ELSE
		bLift_InTarget := FALSE;
	END_IF;

1:	(*IDLE*)
	IF bLift_Start THEN
		bLift_InTarget := FALSE;
		iState_Lift := 2;
	END_IF;

2:	(*MovingToTarget*)
	bLift_InTarget := FALSE;
	IF fLift_TargetPos > fLift_CurrentPos THEN
		(*Moving up*)
		fLift_CurrentPos := fLift_CurrentPos + ABS(fLift_Velo);
	ELSIF fLift_TargetPos < fLift_CurrentPos THEN
		(*Moving down*)
		fLift_CurrentPos := fLift_CurrentPos - ABS(fLift_Velo);
	END_IF;
	(*Limit output*)
	fLift_CurrentPos := LIMIT(-fPOS_MAX_DOWN, fLift_CurrentPos, 10);
	(* Moved close to target*)
	IF (ABS(fLift_CurrentPos - fLift_TargetPos) <= ABS(fLift_Velo) ) THEN
		fLift_CurrentPos := fLift_TargetPos;
		iState_Lift := 3;
	END_IF;
	(*Start has been removed*)
	IF NOT bLift_Start THEN
		iState_Lift := 1;
	END_IF;

3:	(*In target*)
	bLift_InTarget := TRUE;
	IF NOT bLift_Start THEN
		iState_Lift := 1;
	END_IF;

ELSE	(*Error / to Default*)
	iState_Lift := 0;
END_CASE;

fPos_Y := -fLift_CurrentPos;
fBasePos_Y := fPos_Y;	(*Used for animations as base position*)


(*define fixture jaws positions*)
IF bFixture_Close THEN
	fPosJawDiff := 0;
ELSE
	fPosJawDiff := 10;
END_IF;

(*Set sensor values*)
(*Set output values*)
bLimit_Top := (fPos_Y <= 0);
bLimit_Bottom := (fPos_Y >= (fPOS_MAX_DOWN-10));
bHome_Sensor := (fPos_Y <= 5) AND (fPos_Y >= -5);

bFixture_Open := NOT bFixture_Close;
bFixture_Closed := bFixture_Close;

IF bDrillOn THEN
	iRPMCurrent := iRPMCurrent + 100;
ELSE
	iRPMCurrent := iRPMCurrent - 20;
END_IF;
iRPMCurrent := LIMIT(0, iRPMCurrent, iSPINDLE_RPM_MAX);
END_FUNCTION_BLOCK

(* POU Simulation/F_CopyPart, ST *)
FUNCTION F_CopyPart : BOOL
(*Moves part data from part to part*)
VAR_INPUT
END_VAR
VAR_IN_OUT
	stPartFrom : ST_Part;	(*The copied part - From*)
	stPartTo : ST_Part;	(*Where to copy the part*)
END_VAR
VAR
END_VAR
(*Moves part data from part to part*)
stPartTo.bExists := stPartFrom.bExists;
stPartTo.bHasHole := stPartFrom.bHasHole;
stPartTo.posX := stPartFrom.posX;
stPartTo.posY := stPartFrom.posY;

F_CopyPart:=TRUE;
END_FUNCTION

(* POU Simulation/F_MovePartForward, ST *)
FUNCTION F_MovePartForward : BOOL
(*Moves parts forward on conveyour, if possible*)
VAR_INPUT
END_VAR
VAR_IN_OUT
	arrParts : ARRAY [0..10] OF ST_Part;	(*Array of parts*)
END_VAR
VAR
	i : INT;	(*indexer*)
	j : INT;	(*indexer*)
END_VAR
(*Moves parts forward as much there is free places*)
FOR i:= 0 TO 9 DO
	j := i +1;
	IF NOT arrParts[i].bExists THEN
		IF arrParts[j].bExists THEN
			F_CopyPart(arrParts[j], arrParts[i]);
			arrParts[j].bExists := FALSE;
			arrParts[j].bHasHole := FALSE;
		END_IF;
	END_IF;
END_FOR;

F_MovePartForward := TRUE;
END_FUNCTION

(* Visualisation Simulator/Components/VC_Beacon
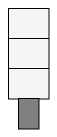
rectangle at (0,0)-(41,31): alarm colour if $red$
rectangle at (0,30)-(41,61): alarm colour if $yellow$
rectangle at (0,60)-(41,91): alarm colour if $green$
1 more shapes without text or variables
*)

(* Visualisation Simulator/ErrorPanels/VC_ErrorDetail_Drill
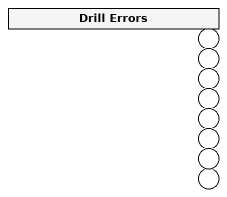
embedded screen at (0,20)-(211,41): VC_ErrorItem
rectangle at (0,0)-(211,21): text "Drill Errors"
embedded screen at (0,40)-(211,61): VC_ErrorItem
embedded screen at (0,160)-(211,181): VC_ErrorItem
embedded screen at (0,60)-(211,81): VC_ErrorItem
embedded screen at (0,80)-(211,101): VC_ErrorItem
embedded screen at (0,100)-(211,121): VC_ErrorItem
embedded screen at (0,120)-(211,141): VC_ErrorItem
embedded screen at (0,140)-(211,161): VC_ErrorItem
*)

(* Visualisation Simulator/ErrorPanels/VC_ErrorDetail_Manip
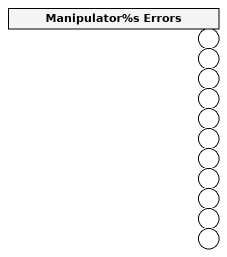
embedded screen at (0,20)-(211,41): VC_ErrorItem
rectangle at (0,0)-(211,21): text "Manipulator%s Errors"; shows $manipName$
embedded screen at (0,40)-(211,61): VC_ErrorItem
embedded screen at (0,60)-(211,81): VC_ErrorItem
embedded screen at (0,80)-(211,101): VC_ErrorItem
embedded screen at (0,80)-(211,101): VC_ErrorItem
embedded screen at (0,100)-(211,121): VC_ErrorItem
embedded screen at (0,120)-(211,141): VC_ErrorItem
embedded screen at (0,140)-(211,161): VC_ErrorItem
embedded screen at (0,160)-(211,181): VC_ErrorItem
embedded screen at (0,180)-(211,201): VC_ErrorItem
embedded screen at (0,200)-(211,221): VC_ErrorItem
embedded screen at (0,220)-(211,241): VC_ErrorItem
*)

(* Visualisation Simulator/VC_ErrorDetails
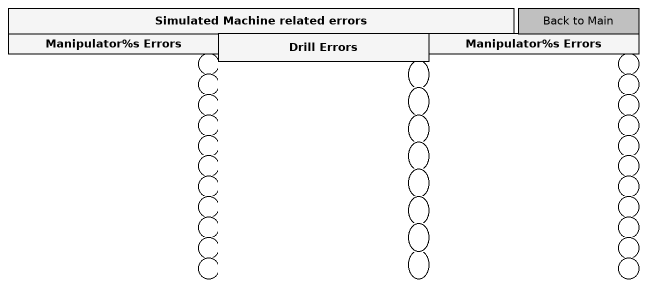
embedded screen at (0,25)-(211,271): VC_ErrorDetail_Manip
rectangle at (0,0)-(506,26): text "Simulated Machine related errors"
embedded screen at (420,25)-(631,271): VC_ErrorDetail_Manip
embedded screen at (210,25)-(421,271): VC_ErrorDetail_Drill
rounded rectangle at (510,0)-(631,26): text "Back to Main"; opens VISU_SimulatedMachine
*)

(* Visualisation Simulator/Components/VC_ErrorItem
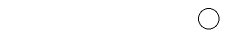
rectangle at (0,0)-(191,21): text "%s :"; shows $name$; alarm colour if $flag$
ellipse at (190,0)-(211,21): alarm colour if $flag$
1 more shapes without text or variables
*)

(* Visualisation Simulator/FBs/VC_FB_Simu_Drill
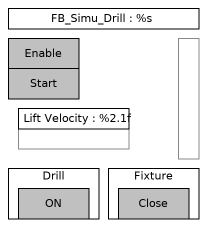
rectangle at (100,160)-(191,211): text "Fixture"
rectangle at (0,160)-(91,211): text "Drill"
rounded rectangle at (0,30)-(71,61): text "Enable"; alarm colour if $FB$.bEnable; toggles $FB$.bEnable
rectangle at (0,0)-(191,21): text "FB_Simu_Drill : %s"; shows $Name$
rounded rectangle at (0,60)-(71,91): text "Start"; alarm colour if $FB$.bLift_Start; taps $FB$.bLift_Start
rectangle at (10,100)-(121,121): text "Lift Velocity : %2.1f"; shows $FB$.fLift_Velo
rounded rectangle at (10,180)-(81,211): text "ON"; alarm colour if $FB$.bDrillOn; toggles $FB$.bDrillOn
rounded rectangle at (110,180)-(181,211): text "Close"; alarm colour if $FB$.bFixture_Close; toggles $FB$.bFixture_Close
2 more shapes without text or variables
1 elements of other kinds (tables, trends, ...) not read
*)

(* Visualisation Simulator/FBs/VC_FB_Simu_Manipulator
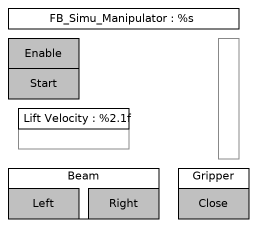
rectangle at (170,160)-(241,211): text "Gripper"
rectangle at (0,160)-(151,211): text "Beam"
rounded rectangle at (0,30)-(71,61): text "Enable"; alarm colour if $FB$.bEnable; toggles $FB$.bEnable
rectangle at (0,0)-(231,21): text "FB_Simu_Manipulator : %s"; shows $Name$
rounded rectangle at (0,60)-(71,91): text "Start"; alarm colour if $FB$.bLift_Start; taps $FB$.bLift_Start
rectangle at (10,100)-(121,121): text "Lift Velocity : %2.1f"; shows $FB$.fLift_Velo
rounded rectangle at (0,180)-(71,211): text "Left"; alarm colour if $FB$.bBeam_Left; toggles $FB$.bBeam_Left
rounded rectangle at (80,180)-(151,211): text "Right"; alarm colour if $FB$.bBeam_Right; toggles $FB$.bBeam_Right
rounded rectangle at (170,180)-(241,211): text "Close"; alarm colour if $FB$.bGripper_Close; toggles $FB$.bGripper_Close
2 more shapes without text or variables
1 elements of other kinds (tables, trends, ...) not read
*)

(* Visualisation Simulator/MachineComponents/VC_Panel_MachineControl
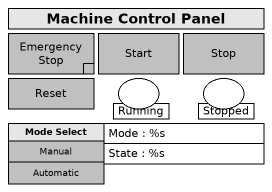
rounded rectangle at (0,25)-(86,66): text "Emergency / Stop"; alarm colour if PRG_Simulator.bBtn_EmergencyStop; toggles PRG_Simulator.bBtn_EmergencyStop
rounded rectangle at (90,25)-(171,66): text "Start"; alarm colour if .I_Btn_Start; taps .I_Btn_Start
rounded rectangle at (0,70)-(86,101): text "Reset"; alarm colour if .I_Btn_Reset; taps .I_Btn_Reset
rounded rectangle at (175,25)-(256,66): text "Stop"; alarm colour if .I_Btn_Stop; taps .I_Btn_Stop
rectangle at (0,0)-(256,21): text "Machine Control Panel"
rectangle at (95,115)-(256,136): text "Mode : %s"; shows .fbStateModel.eMode
rectangle at (95,135)-(256,156): text "State : %s"; shows .fbStateModel.eState
embedded screen at (0,115)-(96,176): VC_Panel_ModeSelector
rectangle at (105,95)-(161,111): text "Running"
rectangle at (190,95)-(246,111): text "Stopped"
ellipse at (110,70)-(151,101): alarm colour if .O_Light_Running
ellipse at (195,70)-(236,101): alarm colour if .O_Light_Stopped
embedded screen at (75,55)-(86,66): VC_sensor
*)

(* Visualisation Simulator/MachineComponents/VC_Panel_MachineControl_simple
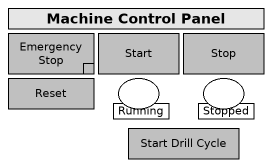
rounded rectangle at (0,25)-(86,66): text "Emergency / Stop"; alarm colour if PRG_Simulator.bBtn_EmergencyStop; toggles PRG_Simulator.bBtn_EmergencyStop
rounded rectangle at (90,25)-(171,66): text "Start"; alarm colour if .I_Btn_Start; taps .I_Btn_Start
rounded rectangle at (0,70)-(86,101): text "Reset"; alarm colour if .I_Btn_Reset; taps .I_Btn_Reset
rounded rectangle at (175,25)-(256,66): text "Stop"; alarm colour if .I_Btn_Stop; taps .I_Btn_Stop
rectangle at (0,0)-(256,21): text "Machine Control Panel"
rectangle at (105,95)-(161,111): text "Running"
rectangle at (190,95)-(246,111): text "Stopped"
ellipse at (110,70)-(151,101): alarm colour if .O_Light_Running
ellipse at (195,70)-(236,101): alarm colour if .O_Light_Stopped
rounded rectangle at (120,120)-(231,151): text "Start Drill Cycle"; alarm colour if .I_Btn_CycleStart; taps .I_Btn_CycleStart
embedded screen at (75,55)-(86,66): VC_sensor
*)

(* Visualisation Simulator/MachineComponents/VC_Panel_ModeSelector
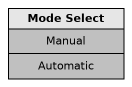
rounded rectangle at (0,20)-(116,46): text "Manual"; alarm colour if .HMI_uModeReq=3; runs INTERN ASSIGN HMI_uModeReq:=(3)
rectangle at (0,0)-(116,21): text "Mode Select"
rounded rectangle at (0,45)-(116,71): text "Automatic"; alarm colour if .HMI_uModeReq=1; runs INTERN ASSIGN HMI_uModeReq:=(1)
*)

(* Visualisation Simulator/Components/VC_Part
rectangle at (0,0)-(41,51): invisible if NOT $part$.bExists
rectangle at (15,0)-(26,41): invisible if NOT $part$.bExists OR NOT $part$.bHasHole
*)

(* Visualisation Simulator/Components/VC_sensor
rectangle at (0,0)-(11,11): alarm colour if $VAR$
*)

(* Visualisation Simulator/MachineComponents/VC_Simu_Conv_In
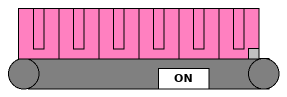
embedded screen at (210,0)-(251,51): VC_Part
embedded screen at (240,40)-(251,51): VC_sensor
embedded screen at (170,0)-(211,51): VC_Part
embedded screen at (130,0)-(171,51): VC_Part
embedded screen at (90,0)-(131,51): VC_Part
embedded screen at (50,0)-(91,51): VC_Part
embedded screen at (10,0)-(51,51): VC_Part
rectangle at (150,60)-(201,81): text "OFF"
rectangle at (150,60)-(201,81): text "ON"; invisible if NOT $MotOn$
3 more shapes without text or variables
*)

(* Visualisation Simulator/MachineComponents/VC_Simu_Drill
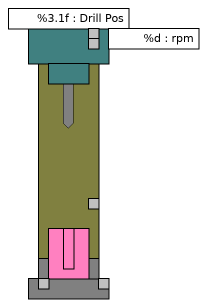
rectangle at (20,20)-(101,56): y offset $FB$.fBasePos_Y
rectangle at (0,0)-(121,21): text "%3.1f : Drill Pos"; shows $FB$.fLift_CurrentPos
embedded screen at (80,20)-(91,31): VC_sensor
embedded screen at (80,190)-(91,201): VC_sensor
embedded screen at (80,30)-(91,41): VC_sensor
polygon at (55,75)-(65,120): alarm colour if $FB$.iRPMCurrent > 0; y offset $FB$.fBasePos_Y
rectangle at (40,55)-(81,76): y offset $FB$.fBasePos_Y
rectangle at (30,250)-(41,271): x offset - $FB$.fPosJawDiff
rectangle at (80,250)-(91,271): x offset $FB$.fPosJawDiff
embedded screen at (40,220)-(81,271): VC_Part
embedded screen at (90,270)-(101,281): VC_sensor
embedded screen at (30,270)-(41,281): VC_sensor
rectangle at (100,20)-(191,41): text "%d : rpm"; shows $FB$.iRPMCurrent
2 more shapes without text or variables
*)

(* Visualisation Simulator/MachineComponents/VC_Simu_Manipulator
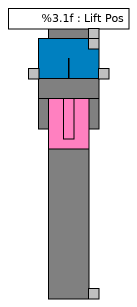
rectangle at (70,40)-(131,81): y offset $FB$.fBasePos_Y
rectangle at (100,60)-(101,81): left $FB$.fPos_Beam_L; right $FB$.fPos_Beam_R; y offset $FB$.fBasePos_Y
rectangle at (70,80)-(131,101): x offset $FB$.fPos_X; y offset $FB$.fBasePos_Y
rectangle at (70,100)-(81,131): x offset $FB$.fPos_X - $FB$.fPosFingerDiff; y offset $FB$.fBasePos_Y
rectangle at (120,100)-(131,131): x offset $FB$.fPos_X + $FB$.fPosFingerDiff; y offset $FB$.fBasePos_Y
embedded screen at (80,100)-(121,151): VC_Part
rectangle at (40,10)-(161,31): text "%3.1f : Lift Pos"; shows $FB$.fLift_CurrentPos
embedded screen at (120,30)-(131,41): VC_sensor
embedded screen at (120,290)-(131,301): VC_sensor
embedded screen at (120,40)-(131,51): VC_sensor
embedded screen at (130,70)-(141,81): VC_sensor
embedded screen at (60,70)-(71,81): VC_sensor
1 more shapes without text or variables
*)

(* Visualisation Simulator/MachineComponents/VC_SimuMach_Controls
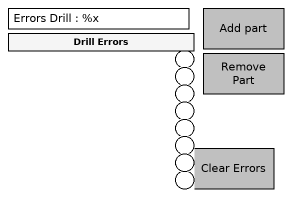
rounded rectangle at (185,140)-(266,181): text "Clear Errors"; alarm colour if PRG_Simulator.bClearErrors; taps PRG_Simulator.bClearErrors
rounded rectangle at (195,45)-(276,86): text "Remove / Part"; alarm colour if PRG_Simulator.bRemovePartFromDrill; taps PRG_Simulator.bRemovePartFromDrill
rectangle at (0,0)-(181,21): text "Errors Drill : %x"; shows PRG_Simulator.wError_Drill; alarm colour if PRG_Simulator.wError_Drill > 0
rounded rectangle at (195,0)-(276,41): text "Add part"; alarm colour if PRG_Simulator.bAddPartInDrill; taps PRG_Simulator.bAddPartInDrill
embedded screen at (0,25)-(186,181): VC_ErrorDetail_Drill
*)

(* Visualisation Simulator/VISU_SimulatedMachine
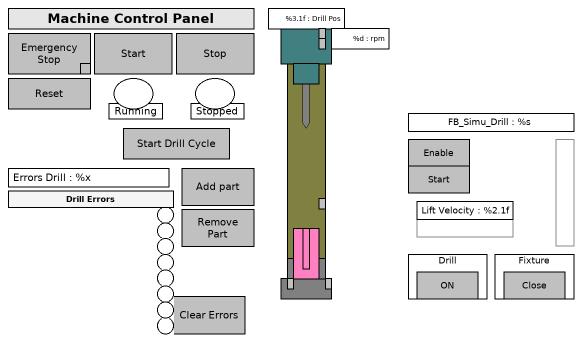
embedded screen at (0,-35)-(246,116): VC_Panel_MachineControl_simple
embedded screen at (260,-35)-(381,256): VC_Simu_Drill
embedded screen at (0,125)-(246,291): VC_SimuMach_Controls
embedded screen at (400,70)-(566,256): VC_FB_Simu_Drill
*)
